	// Confirm Check variables
	fb_ConfirmCheck 		: ARRAY[SorterExample.DIVERTMIN..SorterExample.NUMBEROFDIVERTS] OF FB_ConfirmCheck;
	st_ConfirmItem 			: ARRAY[SorterExample.DIVERTMIN..SorterExample.NUMBEROFDIVERTS] OF ST_Item;
	nConfirmItemIndex 		: UDINT;
	
	BlankItem				: ST_Item := (ID := ''
											, UniqueID := 0
											, Destination := 0
											, Status := E_StatusCode.No_Status
											, ExtStatus := E_StatusCode.No_Status
											, DeviceID := ''
											, MessageType := E_MessageIds.NoMessage_00);

	workingItem			: ST_Item;	// Actual item to induct

	LastItemInducted 	: STRING;
	nIndexToClear		: UDINT;	// Clear Item Array at this index
	nItemArraySize		: UDINT;

	rInductPE			: R_TRIG; 	// Capture the Rising edge of the Induct PE
	fInductPE			: F_TRIG; 	// Capture the Falling edge of the Induct PE
	sMessage			: STRING;

	st_DisplayItem		:st_Item;
	
	LogSorterDump: BOOL := FALSE;
END_VAR

// Initialize FB_ItemExtBuffer
fbSorterDiagLog(st_BufferData := aSorterDiagLog);

(*
// Test visu variables	
inductPE := SorterInductPE;
ItemsOut := Items;
ArrivalOut := ArrivalBuffer;
// End test variables
*)
(*
	Capture the Upper/Lower bound of relevant IO_OUT arrays for looping purposes
	ItemsArrayMax/Min for the sorter array slot count
*)
// Size is Max - Min + 1 to capture both extremes
nItemArraySize := ItemsArrayMax - ItemsArrayMin + 1;

FOR divertIndex := DivertArrayMin TO DivertArrayMax DO
	fb_DivertFullMonitor(Divert := aDiverts[divertIndex]);
END_FOR

(*
	Detect barcode receipt after item is already in Item array
	the tempItem is reset when the induct PE is cleared
	The tempItem is populated when the induct PE is blocked and there
	is not an associated barcode waiting to be inducted
*)
IF st_tempItem.Item.ID <> '' THEN
	// Test the IN_ItemToInduct.ID for a value
	// This record will be cleared as soon as it reaches the sorter loop
	IF In_ItemToInduct.ID <> '' THEN
		// The tempItem is overwritten with the IN_ItemToInduct after it is updated
		// But the starting encoder count is not changed so the same items can be updated
		// if the destination update is received while the item is still being inducted
		IF In_ItemToInduct.ID <> st_tempItem.Item.ID THEN 
			// Set the starting count for the testing/updating process
			// The testEncodeCount is incremented upon start, so we start -1 of the encoder count for the item
			testEncoderCount := f_CalculateIndex(Offset := -1, InitialValue:= st_tempItem.Counts, BufferSize := nItemArraySize);
			// Clear the length and start over
			In_ItemToInduct.Length := 0;
			st_tempItem.Item := In_ItemToInduct;
		END_IF 
		// Test for a change of destination after the barcode data has been received
		IF In_ItemToInduct.Destination <> st_tempItem.Item.Destination THEN 
			// Set the starting count for the testing/updating process
			// The testEncodeCount is incremented upon start, so we start -1 of the encoder count for the item
			testEncoderCount := f_CalculateIndex(Offset := -1, InitialValue:= st_tempItem.Counts, BufferSize := nItemArraySize);
			// Clear the length and start over
			In_ItemToInduct.Length := 0;
			// Copy the IN_ItemToInduct to prevent running this until something else in the record changes
			st_tempItem.Item := IN_ItemToInduct;
		END_IF
	END_IF 
END_IF


// Test for the rising edge of the induct PE
// Use this rising edge to log the IN_ItemToInduct record
rInductPE(CLK:= st_Sorter.InductPE, Q =>);

IF rInductPE.Q THEN
	IF .nSorterLogEnable.SORTER_INDUCT THEN
		sMessage := CONCAT(' Item: ', In_ItemToInduct.ID);
		sMessage := CONCAT(sMessage, ' Pulses: ');
		sMessage := CONCAT(sMessage, UDINT_TO_STRING(st_Sorter.EncoderCounts));
		// Write to the Error List
		ADSLOGSTR( msgCtrlMask := ADSLOG_MSGTYPE_HINT OR ADSLOG_MSGTYPE_LOG
			, msgFmtStr := 'Induct Info: %s'
			, strArg := sMessage);
	END_IF
END_IF
// Test for the falling edge of the induct PE
// Use this falling edge to clear the IN_ItemToInduct record
fInductPE(CLK:= st_Sorter.InductPE, Q =>);

IF fInductPE.Q THEN
	IF .nSorterLogEnable.SORTER_INDUCT THEN
		sMessage := CONCAT(' Item: ', In_ItemToInduct.ID);
		sMessage := CONCAT(sMessage,' Pulses: ');
		sMessage := CONCAT(sMEssage, UDINT_TO_STRING(st_Sorter.EncoderCounts));
		// Write to the Error List
		ADSLOGSTR( msgCtrlMask := ADSLOG_MSGTYPE_HINT OR ADSLOG_MSGTYPE_LOG
			, msgFmtStr := 'Cleared Induct Info: %s'
			, strArg := sMessage);
	END_IF
	// Clear the record
	In_InductingItem :=  BlankItem;
END_IF

// Process every array index between the current index and the last processed index
WHILE st_Sorter.EncoderCounts <> testEncoderCount DO

	// Capture the lastEncoderCount before changing it for comparison of last inducted items
	lastCompareCount := testEncoderCount;

	// Increment the testEncoderCount
	// The testEncoderCount variable will be used throughout the processing to ensure
	//	that all array elements are processed
	testEncoderCount := f_CalculateIndex(Offset := 1, InitialValue:= testEncoderCount, BufferSize := nItemArraySize);
	IF st_Sorter.InductPE THEN
	  	IF (In_ItemToInduct.ID <> '') THEN
			In_InductingItem := In_ItemToInduct;
			In_ItemToInduct := BlankItem;
			IF .nSorterLogEnable.SORTER_INDUCT_PE THEN
				sMessage := CONCAT(' Item: ', In_InductingItem.ID);
				sMessage := CONCAT(sMessage,' Pulses: ');
				sMessage := CONCAT(sMessage, UDINT_TO_STRING(st_Sorter.EncoderCounts));
				sMessage := CONCAT(sMessage,' Dest: ');
				sMessage := CONCAT(sMessage, DINT_TO_STRING(In_InductingItem.Destination));
				// Write to the Error List
				ADSLOGSTR( msgCtrlMask := ADSLOG_MSGTYPE_HINT OR ADSLOG_MSGTYPE_LOG
					, msgFmtStr := 'Inducting Info: %s'
					, strArg := sMessage);
			END_IF
		END_IF
	  	IF (In_InductingItem.ID <> '') THEN
			LastItemInducted := In_InductingItem.ID;
			IF aItems[testEncoderCount].ID <> '' THEN
				IF aItems[testEncoderCount].Status >= E_StatusCode.Diverting AND aItems[testEncoderCount].Status <= E_StatusCode.Divert_UnknownError THEN
					aItems[testEncoderCount].Status := E_StatusCode.Divert_UnknownError;
				END_IF
				UpdateSorterLog(Status := aItems[testEncoderCount].Status, ItemID := aItems[testEncoderCount].UniqueID);
			END_IF
		
			// Set the Item status
			In_InductingItem.Status := E_StatusCode.In_Sorter;

			// Check for destination full on the first pass, then ignore it.
			IF In_InductingItem.Length = 0 THEN
				IF aDiverts[In_InductingItem.DestinationIdx].Full THEN
					IF st_Sorter.Config.RecircUsed THEN
						In_InductingItem.Destination := st_Sorter.Config.RecircDestination;
						In_InductingItem.DestinationIdx := st_Sorter.Config.RecircDestIdx;
						In_InductingItem.ExtStatus := E_StatusCode.Divert_Recirculated;
					ELSE
						In_InductingItem.Destination := st_Sorter.Config.DefaultDestination;
						In_InductingItem.DestinationIdx := st_Sorter.Config.DefaultDestIdx;
						In_InductingItem.ExtStatus := E_StatusCode.Divert_Full;
					END_IF
				END_IF
			END_IF
			// Clear the extend counter
			tailendcount := 0;

			// Copy the ItemToInduct to the WorkingItem that will be inducted
			workingItem := In_InductingItem;
			// Increment the Length on the ItemToInduct record, then it will be added to the array
			//  and the length will increment
			In_InductingItem.Length := In_InductingItem.Length +  1;
			// Determined by UniqueID = 0
		ELSE //If the item makes it to the sorter, but is not identified, induct the item with tempItem.Item
			LastItemInducted := 'UNKNOWN';
			UpdateSorterLog(Status := E_StatusCode.UnidentifiedItem, ItemID := st_tempItem.Item.UniqueID);

			// Process this the first time
			IF st_tempItem.Item.Length = 0 THEN
				IF aDiverts[st_Sorter.Config.DefaultDestIdx].Full THEN
					IF st_Sorter.Config.RecircUsed THEN
						st_tempItem.Item.Destination := st_Sorter.Config.RecircDestination;
						st_tempItem.Item.DestinationIdx := st_Sorter.Config.RecircDestIdx;
						st_tempItem.Item.ExtStatus := E_StatusCode.Divert_Recirculated;
					ELSE
						st_tempItem.Item.Destination := st_Sorter.Config.DefaultDestination;
						st_tempItem.Item.DestinationIdx := st_Sorter.Config.DefaultDestIdx;
						st_tempItem.Item.ExtStatus := E_StatusCode.Divert_Full;
					END_IF
				ELSE
					st_tempItem.Item.Destination := st_Sorter.Config.DefaultDestination;
					st_tempItem.Item.DestinationIdx := st_Sorter.Config.DefaultDestIdx;
				END_IF		
			END_IF
			// Copy the tempItem.Item to the WorkingItem that will be inducted
			workingItem := st_tempItem.Item;
			// Increment the Length on the ItemToInduct record, then it will be added to the array
			//  and the length will increment
			st_tempItem.Item.Length := st_tempItem.Item.Length +  1;
		END_IF

		// Induct everything
		aItems[testEncoderCount] := workingItem;
		fbSorterDiagLog.AddItem(workingItem);
	// Follow this path when the induct photo-eye is cleared
	ELSE
		// Extend the end of the item by a set amount, or to a mimimum length
		// Test to verify that the Item index is clear, and we are still extending the length of the item
		IF aItems[lastCompareCount].ID <> '' THEN
			IF tailendcount < st_Sorter.Config.TailEndLength AND st_Sorter.Config.TailEndLength > 0 THEN
				aItems[testEncoderCount] := aItems[lastCompareCount]; 
				fbSorterDiagLog.AddItem(aItems[lastCompareCount]);
				aItems[testEncoderCount].Length := aItems[testEncoderCount].Length + 1;
				tailendcount := tailendcount + 1;
			END_IF
			IF aItems[lastCompareCount].Length < st_Sorter.Config.MinimumLength AND st_Sorter.Config.MinimumLength > 0 THEN
				aItems[testEncoderCount] := aItems[lastCompareCount]; 
				fbSorterDiagLog.AddItem(aItems[lastCompareCount]);
				aItems[testEncoderCount].Length := aItems[testEncoderCount].Length + 1;
			END_IF
		END_IF
	END_IF
END_WHILE

// Process every array index between the current index and the last processed exit index
WHILE st_Sorter.EncoderCounts <> exitEncoderCount DO

	// Increment the exitEncoderCount
	// The exitEncoderCount variable will be used throughout the processing to ensure
	//	that all array elements are processed
	exitEncoderCount := f_CalculateIndex(Offset := 1, InitialValue:= exitEncoderCount, BufferSize := nItemArraySize);
	// Process the diverts relative to the current encoder count
	FOR divertIndex := DivertArrayMin TO DivertArrayMax DO
		// Get the distance to each divert, distance is the number of pulses to actuation
		Divertoffset := aDiverts[divertIndex].Config.Distance;
		// Calculate the index of the item to test for a divert
		// Subtract the offset from the current encoder count (exitEncoderCount)
		// As the encoder count increases, the current index pointer advances
		// Subtracting looks backwards into the sorter item array to test for items at the diverts
		//	distance that should be diverted
		nTestItemIndex := F_CalculateIndex(initialvalue := exitEncoderCount
										, offset := -(Divertoffset)
										, BufferSize := (ItemsArrayMax + 1));	
		//Setup Out2Item for energizing 2nd divert output
		Output2ItemIndex := F_CalculateIndex(initialvalue := exitEncoderCount
										, offset := -(Divertoffset + UINT_TO_INT(st_Sorter.Config.Output2Offset))
										, BufferSize := (ItemsArrayMax + 1));	
		// Log Diverts
		IF aItems[nTestItemIndex].DestinationIdx = divertIndex THEN
			IF .nSorterLogEnable.SORTER_DIVERTS THEN
				sMessage := CONCAT(' Item: ', aItems[nTestItemIndex].ID);
				sMessage := CONCAT(sMessage,' Index: ');
				sMessage := CONCAT(sMessage, UDINT_TO_STRING(nTestItemIndex));
				sMessage := CONCAT(sMessage,' Dest: ');
				sMessage := CONCAT(sMessage, DINT_TO_STRING(aItems[nTestItemIndex].Destination));
				sMessage := CONCAT(sMessage,' DestIdx: ');
				sMessage := CONCAT(sMessage, DINT_TO_STRING(aItems[nTestItemIndex].DestinationIdx));
				sMessage := CONCAT(sMessage,' Divert Status: ');
				sMessage := CONCAT(sMessage, DINT_TO_STRING(aDiverts[DivertIndex].Status));
				sMessage := CONCAT(sMessage,' Item Status: ');
				sMessage := CONCAT(sMessage, DINT_TO_STRING(aItems[nTestItemIndex].Status));
				// Write to the Error List
				ADSLOGSTR( msgCtrlMask := ADSLOG_MSGTYPE_HINT OR ADSLOG_MSGTYPE_LOG
					, msgFmtStr := 'Item at Divert Index: %s'
					, strArg := sMessage);
			END_IF
		END_IF
		fb_DivertDecision( bLog := .nDivertLogEnable.DIVERT_DECISION 
					 , Output1Item		:= aItems[nTestItemIndex]
					 , Output2Item		:= aItems[Output2ItemIndex]
					 , Divert 			:= aDiverts[DivertIndex]
					 , DivertIndex		:= DivertIndex
					 );
		// Calculate the distance to the confirm PE to test for a successful divert
		nConfirmItemIndex := F_CalculateIndex(initialvalue := exitEncoderCount
										, offset := -(Divertoffset + aDiverts[divertIndex].Config.ConfirmDist)
										, BufferSize := (ItemsArrayMax + 1));
		// Log Confirms
		IF aItems[nConfirmItemIndex].Status = E_StatusCode.Diverting AND aItems[nConfirmItemIndex].UniqueID <> 0 THEN
			IF .nSorterLogEnable.SORTER_CONFIRMS THEN
				sMessage := CONCAT(' Item: ', aItems[nConfirmItemIndex].ID);
				sMessage := CONCAT(sMessage,' Index: ');
				sMessage := CONCAT(sMessage, UDINT_TO_STRING(nConfirmItemIndex));
				sMessage := CONCAT(sMessage,' Dest: ');
				sMessage := CONCAT(sMessage, DINT_TO_STRING(aItems[nConfirmItemIndex].Destination));
				sMessage := CONCAT(sMessage,' DestIdx: ');
				sMessage := CONCAT(sMessage, DINT_TO_STRING(aItems[nConfirmItemIndex].DestinationIdx));
				sMessage := CONCAT(sMessage,' Divert Status: ');
				sMessage := CONCAT(sMessage, DINT_TO_STRING(aDiverts[DivertIndex].Status));
				sMessage := CONCAT(sMessage,' Item Status: ');
				sMessage := CONCAT(sMessage, DINT_TO_STRING(aItems[nTestItemIndex].Status));
				// Write to the Error List
				ADSLOGSTR( msgCtrlMask := ADSLOG_MSGTYPE_HINT OR ADSLOG_MSGTYPE_LOG
					, msgFmtStr := 'Item at Confirm Index: %s'
					, strArg := sMessage);
			END_IF
		END_IF
		fb_ConfirmCheck[divertIndex] ( bLog := .nDivertLogEnable.DIVERT_DECISION 
					 , ConfirmItem		:= aItems[nConfirmItemIndex]
					 , ConfirmPE 		:= aDiverts[DivertIndex].ConfirmPE
					 , DivertIndex		:= DivertIndex
					 , bIsDischarge		:= aDiverts[DivertIndex].Config.IsDischarge
					 , DetectedItem => st_ConfirmItem[DivertIndex]
					 );
	END_FOR
	
	// Capture the last item discharged by this sorter section
	IF st_ConfirmItem[DivertArrayMax].ID <> '' THEN
		st_DischargeItem := st_ConfirmItem[DivertArrayMax];
	END_IF

	// Clear the Item array ahead of the current encoder count
	nIndexToClear := f_CalculateIndex(Offset := 400, InitialValue:= exitEncoderCount, BufferSize := nItemArraySize);
	IF aItems[nIndexToClear].ID <> '' THEN
		IF .nSorterLogEnable.SORTER_DUMP THEN
			sMessage := CONCAT(' Item: ', aItems[nIndexToClear].ID);
			sMessage := CONCAT(sMessage,' Index: ');
			sMessage := CONCAT(sMessage, UDINT_TO_STRING(nIndexToClear));
			sMessage := CONCAT(sMessage,' Item Status: ');
			sMessage := CONCAT(sMessage, DINT_TO_STRING(aItems[nIndexToClear].Status));
			// Write to the Error List
			ADSLOGSTR( msgCtrlMask := ADSLOG_MSGTYPE_HINT OR ADSLOG_MSGTYPE_LOG
				, msgFmtStr := 'Clear Ahead Dump Info: %s'
				, strArg := sMessage);
		END_IF
	END_IF
	aItems[nIndexToClear] := BlankItem;

END_WHILE

END_PROGRAM

// ---- FunctionBlocks/Utils/Events/FB_Intlks_NoLatch.TcPOU
FUNCTION_BLOCK FB_Intlks_NoLatch
(*
=====================================================================
	Copyright ©  Syscon Automation.  All Rights Reserved.
	Version 1 Release 1 2018
=====================================================================
 
	This FB monitors 16 interlock inputs
	Each "Good or OK" State for each Interlock Input is configurable (Default is 0=OK, 1=trip)
	Interlocks may be configured as Bypassable.
 --------------------------------------------------------------------
*)
 
VAR_INPUT
	In_Intlks:	ARRAY[0..15] OF BOOL;		// Interlocks 0 to 15 Input
	CFG_IntlksArry:	ARRAY[0..15] OF ST_CfgEvents;	// Configuration of Interlocks
END_VAR
VAR_OUTPUT
	All_Intlk_OK: BOOL;		// Status Bit Showing that ALL Interlocks are OK to RUN (either interlock is OK or it has been bypassed (0= Interlock Enabled-Stop, 1= OK to Run)	
	STS_Intlks:	ARRAY[0..15] OF ST_EventSts;		// Status of each Interlock State (0= OFF, 1=ON)
	STS_BypassActive: BOOL;		// Status Bit Showing that a Bypass is Active (0= No Active Bypass, 1= A Bypass is Active) 
	
END_VAR
VAR
	Intlk_CrntStsArry:	ARRAY[0..15] OF BOOL;		// The Current state of the interlock after compared to OK state
	Intlks_Bypassed:	ARRAY[0..15] OF BOOL;		// Interlocks where Bypass is ON and Allowed
	Sts_Intlks_BypassNotAllowed:	ARRAY[0..15] OF BOOL;		// Status representing each Non Bypassable Interlock State (0= OFF, 1=ON)
	Intlk_ON:	BOOL;		// Testing Bit to Show that an Interlock is Active Based on Current OK State (ignoring Latches and Bypassing)
	i: INT;		//index
END_VAR

// Run loop to check each input
FOR i := 0 TO 15 DO
	// Compare to OK State
	Intlk_CrntStsArry[i] := In_Intlks[i] XOR CFG_IntlksArry[i].OKState;
		
	//Set Status 
	STS_Intlks[i].Status := Intlk_CrntStsArry[i];
		
	//Look for Bypass State
	Intlks_Bypassed[i] := CFG_IntlksArry[i].ByPssAllwd AND CFG_IntlksArry[i].HMI_BypassPB; 
	Sts_Intlks_BypassNotAllowed[i] := NOT Intlks_Bypassed[i];  
	Sts_Intlks_BypassNotAllowed[i] := Sts_Intlks_BypassNotAllowed[i] AND STS_Intlks[i].Status;
	
	//Update Status based on bypass
	STS_Intlks[i].Status := STS_Intlks[i].Status AND (NOT Intlks_Bypassed[i]);
	STS_Intlks[i].Description := CFG_IntlksArry[i].Description;
	STS_Intlks[i].DeviceLabel := CFG_IntlksArry[i].DeviceLabel;
	IF STS_Intlks[i].Status AND STS_Intlks[i].Description <> '' THEN
		STS_Intlks[i].StatusTxt := 'TRUE';
	ELSE
		STS_Intlks[i].StatusTxt := 'FALSE';
	END_IF
END_FOR

//Set Up test bit showing all active interlocks ignoring bypasses and latching
Intlk_ON := In_Intlks[0] OR In_Intlks[1] OR In_Intlks[2] OR In_Intlks[3] 
			OR In_Intlks[4]OR In_Intlks[5] OR In_Intlks[6] OR In_Intlks[7]
			OR In_Intlks[8] OR In_Intlks[9] OR In_Intlks[10] OR In_Intlks[11]
			OR In_Intlks[12] OR In_Intlks[13] OR In_Intlks[14] OR In_Intlks[15];
						
// Set up bit showing that a bypass is active			
STS_BypassActive := Intlks_Bypassed[0] OR Intlks_Bypassed[1] OR Intlks_Bypassed[2] OR Intlks_Bypassed[3]
			OR Intlks_Bypassed[4] OR Intlks_Bypassed[5] OR Intlks_Bypassed[6] OR Intlks_Bypassed[7]
			OR Intlks_Bypassed[8] OR Intlks_Bypassed[9] OR Intlks_Bypassed[10] OR Intlks_Bypassed[11]
			OR Intlks_Bypassed[12] OR Intlks_Bypassed[13] OR Intlks_Bypassed[14] OR Intlks_Bypassed[15];
			
// Set up bit showing that All interlocks are good			
All_Intlk_OK := NOT( STS_Intlks[0].Status OR STS_Intlks[1].Status OR STS_Intlks[2].Status OR STS_Intlks[3].Status
			OR STS_Intlks[4].Status OR STS_Intlks[5].Status OR STS_Intlks[6].Status OR STS_Intlks[7].Status
			OR STS_Intlks[8].Status OR STS_Intlks[9].Status OR STS_Intlks[10].Status OR STS_Intlks[11].Status
			OR STS_Intlks[12].Status OR STS_Intlks[13].Status OR STS_Intlks[14].Status OR STS_Intlks[15].Status);

END_FUNCTION_BLOCK

// ---- FunctionBlocks/Utils/FB_FlipFlop.TcPOU
(*
Function Block to create a flip flop output based on a single input trigger.
Each transition of In from Low to High will chnage Out output state to change
*)
FUNCTION_BLOCK FB_FlipFlop

VAR_INPUT
	In:	BOOL;
END_VAR
VAR_OUTPUT
	Out:	BOOL;
END_VAR
VAR

	In_rtrig: R_TRIG;
END_VAR

// Input Trigger
In_rtrig(CLK:=In);

// Cpntroll Output
IF In_rtrig.Q AND NOT Out THEN
	Out := TRUE;
ELSIF In_rtrig.Q AND Out THEN
	Out := FALSE;
END_IF

END_FUNCTION_BLOCK

// ---- FunctionBlocks/Utils/Filters/FB_DigDebnce_Off.TcPOU
(*
Function Block to filter the OFF of a digital input In
The normal OK state can be configured with CFG_OKState
The Time for the Off delay is configured by CFG_OffDlyTime
and can be simulated using the In_Sim input
If the input In goes true
If the input In goes false the output CFG_OffDlyTime will be held on until the off delay time has elapsed
The status output Sts_OffDlyActive shows that the delay is active
*)
FUNCTION_BLOCK FB_DigDebnce_Off
VAR_INPUT
	In:	BOOL;	// Digital Input
	CFG_OKState:	BOOL;		// The OK or ON State of the Input (0 or 1)
	CFG_OffDlyTime:	TIME;		// Time to delay Output turning Off after Input is Off
	In_Sim:	BOOL;		// Simulation Input Bit acts just like the input but can be forced from the program for testing
END_VAR
VAR_OUTPUT
	Out:	BOOL;		// Output Based on ON or OK state
	OutOffFltrd:	BOOL;		// Off filtered Only OutPut
	Sts_OffDlyActive: BOOL;
END_VAR
VAR
	OffDlyTof: TOF;
	
END_VAR

// Compare to normal ON state
Out := (In OR In_Sim) XOR CFG_OKState;

//Setup Off Delay
OffDlyTof(IN:= Out , PT:= CFG_OffDlyTime , Q=> OutOffFltrd , ET=> );
Sts_OffDlyActive := Out <> OutOffFltrd;

END_FUNCTION_BLOCK

// ---- FunctionBlocks/Utils/Filters/FB_DigDebnce_On.TcPOU
(*
Function Block to filter the ON of a digital input In
The normal OK state can be configured with CFG_OKState
The Time for the On delay is configured by CFG_OnDlyTime
and can be simulated using the In_Sim input
If the input In goes true the output OutOnFltrd is set to true after the on delay time has elapsed
If the input In goes false the output will go False
The status output Sts_OnDlyActive shows that the delay is active

*)
FUNCTION_BLOCK FB_DigDebnce_On
VAR_INPUT
	In:	BOOL;	// Digital Input
	CFG_OKState:	BOOL;		// The OK or ON State of the Input (0 or 1)
	CFG_OnDlyTime:	TIME;		// Time to delay Output turning On after Input is On
	In_Sim:	BOOL;		// Simulation Input Bit acts just like the input but can be forced from the program for testing
END_VAR
VAR_OUTPUT
	Out:	BOOL;		// Output Based on ON or OK state
	OutOnFltrd:	BOOL;		// ON filtered Only Output 
	Sts_OnDlyActive: BOOL;
	
END_VAR
VAR
	OnDly_Ton: TON;
	
	
END_VAR

// Compare to normal ON state
Out := (In OR In_Sim) XOR CFG_OKState;

// Setup On Delay
OnDly_Ton(IN:= Out, PT:= CFG_OnDlyTime , Q=> OutOnFltrd , ET=> );
Sts_OnDlyActive := Out <> OutOnFltrd;

END_FUNCTION_BLOCK

// ---- FunctionBlocks/Utils/Filters/F_Clip.TcPOU
(*
Function to clip the input InX within the range of InMax and InMin
the additional outputs show if the input is actively beig clipped

*)
FUNCTION F_Clip : INT
VAR_INPUT
	InX:	INT;
	InMax:	INT;
	InMin:	INT;
END_VAR
VAR_OUTPUT
	MaxClipActive:	BOOL;
	MinClipActive:	BOOL;
END_VAR
VAR
END_VAR

IF InX > InMAx THEN 
	MaxClipActive := TRUE;
	MinClipActive := FALSE;
	F_Clip:= InMax;
ELSIF InX < InMin THEN 
	MaxClipActive := FALSE;
	MinClipActive := TRUE;
	F_Clip:= InMin;
ELSE
	MaxClipActive := FALSE;
	MinClipActive := FALSE;
	F_Clip:= InX;
END_IF

END_FUNCTION

// ---- FunctionBlocks/Utils/F_DecIndex.TcPOU
FUNCTION F_DecIndex : INT
VAR_INPUT
	IDX:	INT;		// Index to be incremented
	IdxMIN:	INT;		// Min Value for index	
	IdxMAX:	INT;		// Max Value for index
END_VAR
VAR
END_VAR

IF IDX > IdxMIN THEN
	F_DecIndex := IDX - 1; 
ELSIF IDX = IdxMIN THEN
	F_DecIndex := IdxMAX;
ELSIF IDX < IdxMIN OR IDX > IdxMAX THEN
	F_DecIndex := IdxMAX;
END_IF

END_FUNCTION

// ---- FunctionBlocks/Utils/SystemCntrl_Example.TcPOU
PROGRAM SystemCntrl_Example
VAR
	dummy_Reset			:	BOOL;
	dummy_Auto			:	BOOL;
	dummy_Stop			:	BOOL;
	Cnvyr_Reset AT %Q*:	BOOL;		// Bit to send to all conveyors to reset faults, safeties and etc
	Cnvyr_Start AT %Q*:	BOOL;		// Bit to send to all conveyors to transition to AUTO
	Cnvyr_Stop AT %Q*:	BOOL;		// Bit to send to all conveyors to Stop/transition to manual and stop

	SysStateCntrlSts		: 	ST_EquipmentStatus;	// System State/Control/Status Data
	SysState				:	FB_SystemCntrl;
	SysStateCntrl_StatePB		:	ST_StateCntrlPB;
	SysIntlksAllOk AT %Q*	:	BOOL;	// Bit to show that System interlocks are OK	
	
	SysEventsArry: ARRAY [0..15] OF BOOL;
	SysEventsAllOk AT %Q*: BOOL;	// Bit to show that Syetem events are all OK If system events are needed use event manager FB tie to here

	
END_VAR

VAR PERSISTENT
	{attribute 'OPC.UA.DA' := '1'}
	cfgSysStateIntlksArry: ARRAY [0..15] OF ST_CfgEvents;
	{attribute 'OPC.UA.DA' := '1'}
	cfgSysStateEvntsArry: ARRAY [0..15] OF ST_CfgEvents;
END_VAR

// Only the Reset function is required in the SystemCntrl Function Block
SysStateCntrl_StatePB.ResetPB := dummy_Reset; 	// All I/O used for a reset, e.g. HMI, push buttons
SysStateCntrl_StatePB.AutoPB := dummy_Auto; 	// All I/O used for a Start, e.g. HMI, push buttons
SysStateCntrl_StatePB.StopPB := dummy_Stop;		// All I/O used for a Stop, e.g. HMI, push buttons

// Set up System Interlocks
(*
SysState.In_SystemIntlks.0 := GVL_IO.SystemAirPressure;
*)

// Setup the InterlockArray since persistent data items cannot by initilaized the same
// Index 0
(*
cfgSysStateIntlksArry[0].Description := 'System Air Pressure';
cfgSysStateIntlksArry[0].DeviceLabel := 'PS22121';
cfgSysStateIntlksArry[0].OKState := TRUE;
*)

// Set up System Events
(*
SysState.In_SystemEvents.0 := SystemSafety.Safety_PanelEstop;
SysState.In_SystemEvents.1 := SystemSafety.Safety_SortArea_PC;
SysState.In_SystemEvents.2 := SystemSafety.Safety_OCRArea_PC;
SysState.In_SystemEvents.3 := SystemSafety.OCR_State.OCREstopOK;
SysState.In_SystemEvents.4 := SystemSafety.OCR_State.OCRDoorOpenOK;
*)
// Setup the EventArray since persistent data items cannot by initilaized the same
// Index 0
cfgSysStateEvntsArry[0].Description := 'Panel E-Stop';
cfgSysStateEvntsArry[0].DeviceLabel := 'PB1';
cfgSysStateEvntsArry[0].OKState := TRUE;
cfgSysStateEvntsArry[0].StopCode := E_StopCodes.SystemStop;
// Index 1
cfgSysStateEvntsArry[1].Description := 'Sort Area Pull Cord';
cfgSysStateEvntsArry[1].DeviceLabel := 'PC1-2';
cfgSysStateEvntsArry[1].OKState := TRUE;
cfgSysStateEvntsArry[1].StopCode := E_StopCodes.SystemStop;
// Index 2
cfgSysStateEvntsArry[2].Description := 'OCR Area Pull Cord';
cfgSysStateEvntsArry[2].DeviceLabel := 'PC3-4';
cfgSysStateEvntsArry[2].OKState := TRUE;
cfgSysStateEvntsArry[2].StopCode := E_StopCodes.SystemStop;
// Index 3
cfgSysStateEvntsArry[3].Description := 'OCR E-Stop';
cfgSysStateEvntsArry[3].DeviceLabel := 'OCRE-Stop';
cfgSysStateEvntsArry[3].OKState := TRUE;
cfgSysStateEvntsArry[3].StopCode := E_StopCodes.SystemStop;
// Index 4
cfgSysStateEvntsArry[4].Description := 'OCR Doop Open';
cfgSysStateEvntsArry[4].DeviceLabel := 'OCRDoor';
cfgSysStateEvntsArry[4].OKState := TRUE;
cfgSysStateEvntsArry[4].StopCode := E_StopCodes.SystemStop;

// Function Call
SysState(
	In_p_EquipStatePB:= SysStateCntrl_StatePB, 
	Cfg_EquipLabel := 'Equip Desc',
	Cfg_EquipIntlksArry:= cfgSysStateIntlksArry,
	Cfg_EquipEvntsArry:= cfgSysStateEvntsArry, 
	Sts_EquipState := SysStateCntrlSts,
);

SysIntlksAllOk := SysState.Sts_All_Intlks_OK;
SysEventsAllOk :=  NOT SysState.Sts_FaultActive;

Cnvyr_Reset := SysState.Out_Reset;
Cnvyr_Start  := SysState.Out_Auto;
Cnvyr_Stop  := SysState.Out_Stop;

END_PROGRAM

// ---- FunctionBlocks/Sorter/VISUs/ArrayInspection.TcVIS
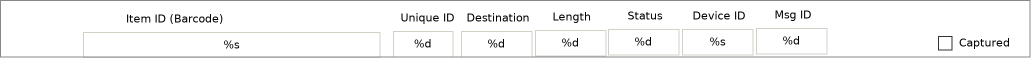
VISUALIZATION ArrayInspection  // 1031x58
VAR_IN_OUT
	st_ItemExt_Disp	:		ST_ItemExt;
(*	ID : STRING := '';		// Bar Code 	
	UniqueID : DINT := 0;		// Generic ID for tracking
	Destination : DINT := 0;
	Length : DINT := 0;
	Status : E_StatusCode := E_StatusCode.No_Status;
	CapturedInMetrics : BOOL;
	DeviceID:	STRING(5);	// Device ID associated with this record
	MessageType:	E_MessageIds;	// Message Type associated with this record
E*)
END_VAR
    Textfield (83,32 297x26), "%s", text variable: st_ItemExt_Disp.ID
    Label (86,11 178x16), "Item ID (Barcode)", invisible if: D
    Label (396,10 63x16), "Unique ID", invisible if: D
    Textfield (393,31 60x26), "%d", text variable: st_ItemExt_Disp.UniqueID
    Label (464,10 68x16), "Destination", invisible if: D
    Textfield (461,31 71x26), "%d", text variable: st_ItemExt_Disp.Destination
    Label (538,9 68x16), "Length", invisible if: D
    Textfield (535,30 71x26), "%d", text variable: st_ItemExt_Disp.Length
    Label (611,8 68x16), "Status", invisible if: D
    Textfield (608,29 71x26), "%d", text variable: st_ItemExt_Disp.Status
    Checkbox (936,28 95x30), "Captured", variable: st_ItemExt_Disp.CapturedInMetrics
    Textfield (682,29 71x26), "%s", text variable: st_ItemExt_Disp.DeviceID
    Label (685,8 68x16), "Device ID", invisible if: D
    Textfield (756,28 71x26), "%d", text variable: st_ItemExt_Disp.MessageType
    Label (759,7 68x16), "Msg ID", invisible if: D
END_VISUALIZATION

// ---- FunctionBlocks/Sorter/VISUs/DiverterTest.TcVIS
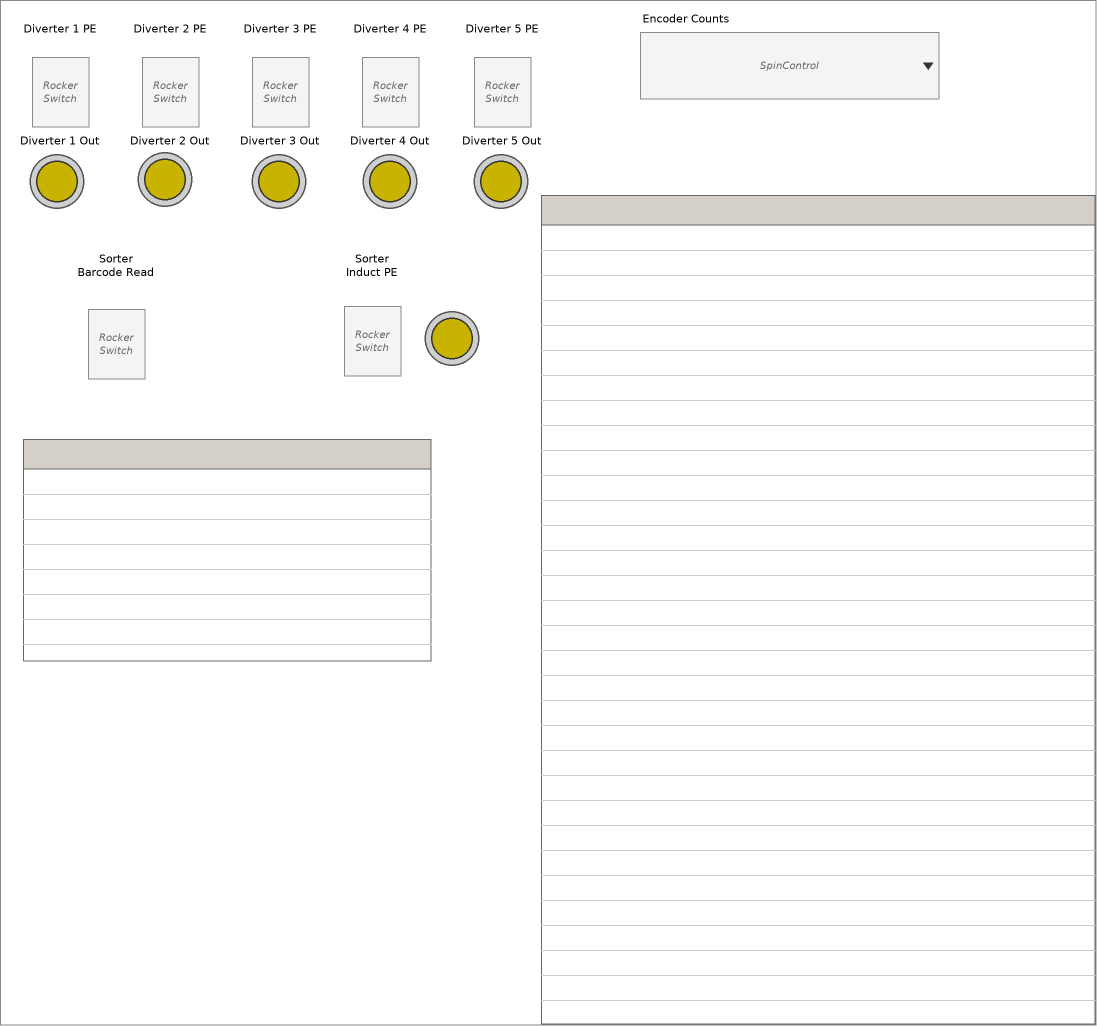
VISUALIZATION DiverterTest  // 1097x1026
    RockerSwitch (32,57 57x70), variable: Diverts[1].JamPE, behaviour: TOGGLE, style: Switch-RockerSwitch-Blue
    Label (9,10 102x38), "Diverter 1 PE"
    RockerSwitch (142,57 57x70), variable: Diverts[2].JamPE, behaviour: TOGGLE, style: Switch-RockerSwitch-Blue
    Label (119,10 102x38), "Diverter 2 PE"
    RockerSwitch (252,57 57x70), variable: Diverts[3].JamPE, behaviour: TOGGLE, style: Switch-RockerSwitch-Blue
    Label (229,10 102x38), "Diverter 3 PE"
    RockerSwitch (362,57 57x70), variable: Diverts[4].JamPE, behaviour: TOGGLE, style: Switch-RockerSwitch-Blue
    Label (339,10 102x38), "Diverter 4 PE"
    RockerSwitch (474,57 57x70), variable: Diverts[5].JamPE, behaviour: TOGGLE, style: Switch-RockerSwitch-Blue
    Label (451,10 102x38), "Diverter 5 PE"
    RockerSwitch (88,309 57x70), variable: BarcodeRead, behaviour: TOGGLE, style: Switch-RockerSwitch-Blue
    Label (65,231 102x69), "Sorter Barcode Read"
    SpinControl (640,32 299x67), variable: MAIN.Sorter1.CurrentRead
    Lamp1 (25,150 64x63), variable: Diverts[1].Output1, style: Lamp-Lamp1-Yellow
    Lamp1 (133,148 64x63), variable: Diverts[2].Output1, style: Lamp-Lamp1-Yellow
    Lamp1 (247,150 64x63), variable: Diverts[3].Output1, style: Lamp-Lamp1-Yellow
    Lamp1 (358,150 64x63), variable: Diverts[4].Output1, style: Lamp-Lamp1-Yellow
    Lamp1 (469,150 64x63), variable: Diverts[5].Output1, style: Lamp-Lamp1-Yellow
    RockerSwitch (344,306 57x70), variable: SorterinductPE, behaviour: TOGGLE, style: Switch-RockerSwitch-Blue
    Label (321,231 102x69), "Sorter Induct PE"
    Lamp1 (420,307 64x63), variable: SorterinductPE, style: Lamp-Lamp1-Yellow
    Table (541,195 554x829), data array: MAIN.aSorterItems
        p3854506369: MAIN.aSorterItems[INDEX].ID
        p2232123230: MAIN.SorterItems[INDEX].ID
        p511219082: MAIN.SorterItems[INDEX].UniqueID
        p1892666644: MAIN.aSorterItems[INDEX].UniqueID
        p1755163831: MAIN.SorterItems[INDEX].Destination
        p338671338: MAIN.aSorterItems[INDEX].Destination
        p4092479075: MAIN.SorterItems[INDEX].Status
        p2170511999: MAIN.aSorterItems[INDEX].Status
        p3723444502: MAIN.aSorterItems[INDEX].CapturedInMetrics
        p2237128397: MAIN.SorterItems[INDEX].CapturedInMetrics
    Table (23,439 408x222), data array: ArrivalOut
        p1755163831: ArrivalOut[INDEX].Destination
        p4092479075: ArrivalOut[INDEX].Status
        p2232123230: ArrivalOut[INDEX].UniqueID
        p511219082: ArrivalOut[INDEX].ID
    Label (9,122 102x38), "Diverter 1 Out"
    Label (119,122 102x38), "Diverter 2 Out"
    Label (229,122 102x38), "Diverter 3 Out"
    Label (339,122 102x38), "Diverter 4 Out"
    Label (451,122 102x38), "Diverter 5 Out"
    Label (635,0 102x38), "Encoder Counts"
END_VISUALIZATION

// ---- FunctionBlocks/Sorter/VISUs/SorterArray.TcVIS
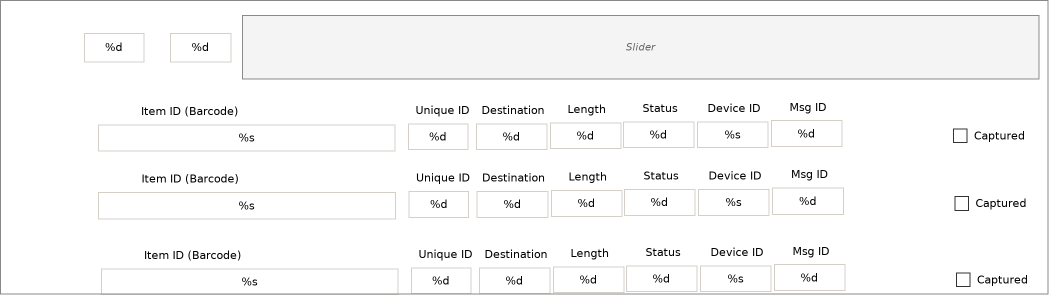
VISUALIZATION SorterArray  // 1049x295
    Frame (15,92 1031x59)
        shows ArrayInspection(st_ItemExt_Disp := MAIN.st_DisplayItem)
        shows ArrayInspection()
        shows ArrayInspection()
    Textfield (170,33 61x29), "%d", text variable: MAIN.nDisplayItemIndex
        OnMouseDown: write MAIN.nDisplayItemIndex via Edit
    Slider (242,15 797x64), variable: MAIN.nDisplayItemIndex, scale 0..100
    Textfield (84,33 60x29), "%d", text variable: MAIN.st_SorterEncoder.CurrentCount
    Frame (15,159 1033x60)
        shows ArrayInspection(st_ItemExt_Disp := ProcessBuffers.st_DisplayItem)
    Frame (18,236 1031x59)
        shows ArrayInspection(st_ItemExt_Disp := SorterProgram.st_DisplayItem)
END_VISUALIZATION

// ---- GlobalTextList.TcGTLO
TEXTLIST GlobalTextList
  645 = '%d'
  572 = '%s'
  787 = 'Captured'
  26 = 'Destination'
  290 = 'Device ID'
  976 = 'Diverter 1 Out'
  64 = 'Diverter 1 PE'
  977 = 'Diverter 2 Out'
  65 = 'Diverter 2 PE'
  978 = 'Diverter 3 Out'
  422 = 'Diverter 3 PE'
  979 = 'Diverter 4 Out'
  423 = 'Diverter 4 PE'
  980 = 'Diverter 5 Out'
  424 = 'Diverter 5 PE'
  950 = 'Encoder Counts'
  341 = 'Item ID (Barcode)'
  534 = 'Length'
  612 = 'Msg ID'
  425 = 'Sorter\n Barcode Read'
  426 = 'Sorter\nInduct PE'
  825 = 'Status'
  666 = 'Unique ID'
END_TEXTLIST
